# EPICS autosave request: slsDetectorApp/Db/slsDetector_settings.req
$(P)$(R)Setting
$(P)$(R)BeamEnergy
$(P)$(R)ThresholdEnergy
$(P)$(R)Trimbits
$(P)$(R)BitDepth
$(P)$(R)TimingMode
$(P)$(R)ReceiverMode
$(P)$(R)ReceiverStream
$(P)$(R)HighVoltage
$(P)$(R)DelayTime
$(P)$(R)NumGates
$(P)$(R)NumCycles
$(P)$(R)NumFrames
$(P)$(R)SetupFile
$(P)$(R)Gate1Width
$(P)$(R)Gate2Width
$(P)$(R)Gate3Width
$(P)$(R)Gate1Delay
$(P)$(R)Gate2Delay
$(P)$(R)Gate3Delay
$(P)$(R)Counter1Threshold
$(P)$(R)Counter2Threshold
$(P)$(R)Counter3Threshold
$(P)$(R)CounterMask
file "ADBase_settings.req", P=$(P), R=$(R)
file "NDFile_settings.req", P=$(P), R=$(R)
